// TwinCAT 3 PLC project OEF_5
// ProgramVersion: 3.1.4024.0
// libraries:
//   Tc2_BABasic, * (Beckhoff Automation GmbH)
//   Tc2_Standard, * (Beckhoff Automation GmbH)
//   Tc2_System, * (Beckhoff Automation GmbH)
//   Tc3_Module, * (Beckhoff Automation GmbH)
// project tree:
//   / PlcTask.TcTTO
//   POUs/ MAIN.TcPOU
// (motion and I/O tree: see PLC project oef_1)
// real-time tasks:
//   TASK PlcTask: cycle T#10ms, priority 20, ADS port 350
//   TASK PlcTask1: cycle T#10ms, priority 21, ADS port 351
//   TASK PlcTask2: cycle T#10ms, priority 22, ADS port 352
//   TASK PlcTask3: cycle T#10ms, priority 23, ADS port 353
//   TASK PlcTask4: cycle T#10ms, priority 24, ADS port 354
// variable links:
//   OEF_5/OEF_5 Instance <-> Device 1 (EtherCAT)/Term 1 (EK1200)/Term 4 (EL3062)
//     PlcTask Inputs/MAIN.Ninput <-> AI Standard Channel 1/Value
//   OEF_5/OEF_5 Instance <-> Device 1 (EtherCAT)/Term 1 (EK1200)/Term 5 (EL4002)
//     PlcTask Outputs/MAIN.Noutput <-> AO Outputs Channel 1/Analog output

CONFIGURATION OEF_5
    RESOURCE PLC ON TwinCAT3
        TASK PlcTask(INTERVAL := T#10ms, PRIORITY := 24);
        PROGRAM MAIN WITH PlcTask : MAIN;
    END_RESOURCE
END_CONFIGURATION

// ---- POUs/MAIN.TcPOU
PROGRAM MAIN
VAR
	Noutput AT %Q*: INT := 0;
	Ninput AT %I*: INT := 0;
	buffer AT %Q*: INT := 0;
END_VAR

buffer := LREAL_TO_INT (F_Scale(Ninput,0,32767,0,100));
Noutput :=LREAL_TO_INT (F_Scale(buffer,-100,2000,0,32767));

END_PROGRAM
